// TIA Portal project "FactoryIO_Template_S7-1200_V16_V16" (V16)
// Vorlageprojekt für das Buch mit Zielsystem S7-1200

(* hardware
DEVICE "S7-1200-Station_1"  S7-1200 Station
   slot 0: "Baugruppenträger_0"  Rack  V1.0
   slot 1: "PLC_1"  CPU 1211C DC/DC/DC  6ES7 211-1AE40-0XB0  V4.1
*)

// ===== PLC "PLC_1"  CPU 1211C DC/DC/DC =====

VAR_GLOBAL   // PLC tag table "Standard-Variablentabelle"
   "fill valve" AT %A0.0 : Bool;
   "start" AT %E0.0 : Bool;
   "stop" AT %E0.1 : Bool;
   "Tag_4" AT %I10.0 : Bool;
   "Tag_5" AT %Q10.0 : Bool;
   "Tag_6" AT %I10.1 : Bool;
   "x" AT %M0.0 : Bool;
   "conveyor" AT %Q0.1 : Bool;
   "t1(1)" AT %M0.1 : Bool;
   "axis sensor" AT %I0.3 : Bool;
   "n" AT %M0.2 : Bool;
   "two axis pick and place 1 z" AT %Q0.2 : Bool;
   "diffuse sensor(1)" AT %I0.2 : Bool;
   "t2(1)" AT %M0.3 : Bool;
   "t2(2)" AT %M0.4 : Bool;
   "tank discharge" AT %Q0.3 : Bool;
   "Tag_1" AT %M0.5 : Bool;
   "t3(1)" AT %M0.6 : Bool;
   "n edge" AT %M0.7 : Bool;
   "t4(1)" AT %M1.0 : Bool;
END_VAR

// folder: System blocks/Program resources

DATA_BLOCK "T1"   // DB1
{ S7_Optimized_Access := 'TRUE' }
AUTHOR : Simatic
FAMILY : IEC
NAME : IEC_TMR
VERSION : 1.0
// stored: InstanceOfName IEC_TIMER
"IEC_TIMER"
BEGIN
END_DATA_BLOCK

DATA_BLOCK "T2"   // DB2
{ S7_Optimized_Access := 'TRUE' }
AUTHOR : Simatic
FAMILY : IEC
NAME : IEC_TMR
VERSION : 1.0
// stored: InstanceOfName IEC_TIMER
"IEC_TIMER"
BEGIN
END_DATA_BLOCK

DATA_BLOCK "T3"   // DB3
{ S7_Optimized_Access := 'TRUE' }
AUTHOR : Simatic
FAMILY : IEC
NAME : IEC_TMR
VERSION : 1.0
// stored: InstanceOfName IEC_TIMER
"IEC_TIMER"
BEGIN
END_DATA_BLOCK

DATA_BLOCK "T4"   // DB4
{ S7_Optimized_Access := 'TRUE' }
AUTHOR : Simatic
FAMILY : IEC
NAME : IEC_TMR
VERSION : 1.0
// stored: InstanceOfName IEC_TIMER
"IEC_TIMER"
BEGIN
END_DATA_BLOCK

// folder: (top level)

FUNCTION "MHJ-PLC-Lab-Function-S71200" : Void   // FC9000, SCL
{ S7_Optimized_Access := 'TRUE' }
VERSION : 0.1
   VAR_TEMP
      rdTimeReturn : Int;
      outputTime : DTL;
      SyncVal : Byte;
      forVal : Int;
      forVal_2 : Int;
      Value : Byte;
   END_VAR
   VAR CONSTANT
      CompVal : Byte := 16#34;
      Value_01 : Byte := 16#11;
      Value_01_DW : DWord := 16#A165_D992;
      Value_02_DW : DWord := 16#58BE_4401;
   END_VAR
BEGIN

   #Value:=PEEK(area := 16#82,
        dbNumber := 0,
        byteOffset := 511);
   #Value := #Value + 1;

   POKE(area := 16#82,
        dbNumber := 0,
        byteOffset := 511,
        value := #Value);

   POKE(area:=16#81,
        dbNumber:=0,
        byteOffset:=1016,
        value:=#Value_01_DW);
   POKE(area := 16#81,
        dbNumber := 0,
        byteOffset := 1020,
        value := #Value_02_DW);

   POKE(area := 16#81,
        dbNumber := 0,
        byteOffset := 511,
        value := B#16#00);

   FOR #forVal := 0 TO 120 DO
       FOR #forVal_2:=0 TO 10 DO
           #rdTimeReturn:=RD_SYS_T(#outputTime);
           #rdTimeReturn := WR_SYS_T(#outputTime);
           #rdTimeReturn := RD_SYS_T(#outputTime);
           #rdTimeReturn := WR_SYS_T(#outputTime);
       END_FOR;
       #SyncVal:= PEEK(area := 16#81,
                      dbNumber := 0,
                      byteOffset := 511);
       IF #SyncVal = #CompVal THEN
          GOTO M_1;
       END_IF;
   END_FOR;
   RETURN;

   M_1:
   POKE(area := 16#81,
        dbNumber := 0,
        byteOffset := 511,
        value := B#16#0);
END_FUNCTION

ORGANIZATION_BLOCK "Main"   // OB1, LAD, ProgramCycle
TITLE = "Main Program Sweep (Cycle)"
{ S7_Optimized_Access := 'TRUE' }
VERSION : 0.1
   VAR_INPUT
      Initial_Call : Bool;   // Initial call of this OB
      Remanence : Bool;   // =True, if remanent data are available
   END_VAR
   VAR_TEMP   // added for the SCL form of the ladder/FBD networks
      _w1 : Bool;
   END_VAR
BEGIN

REGION Network 1: Konnektierungsbaustein für PLC-Lab
   // Im Netzwerk 1 wird der Konnektierungsbaustein für PLC-Lab aufgerufen.
   // Dieser Aufruf darf nicht entfernt werden!
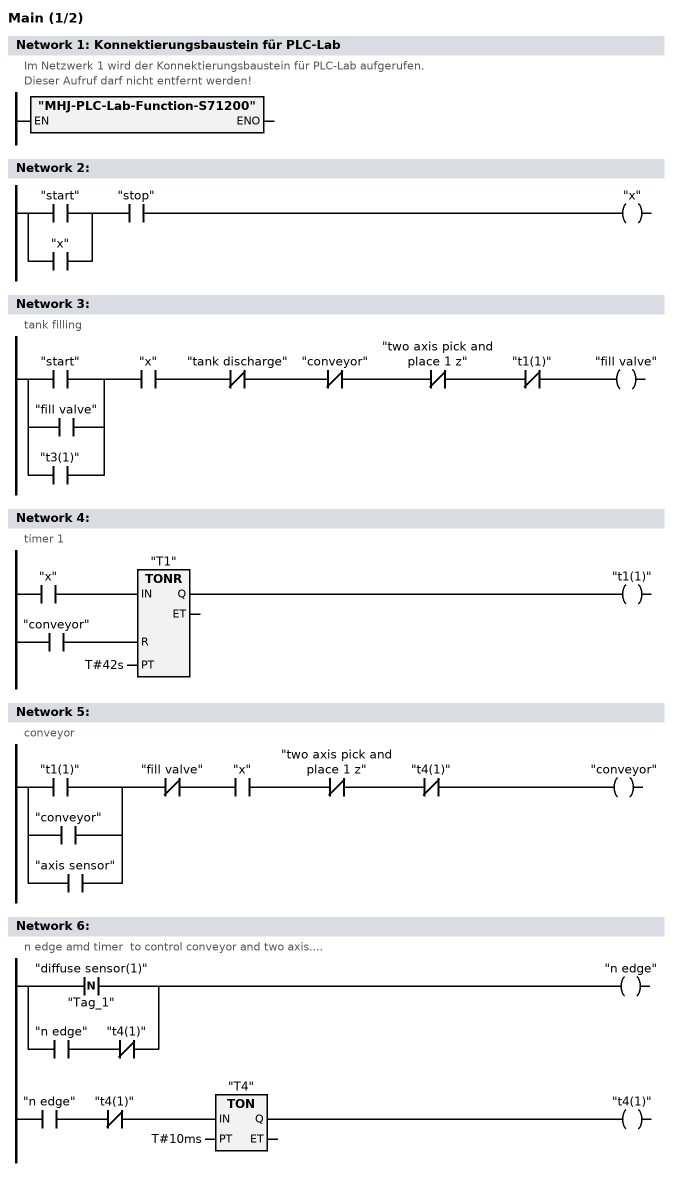
   RUNG wire#powerrail
      "MHJ-PLC-Lab-Function-S71200"()
   END_RUNG
   // the same network as SCL:
   "MHJ-PLC-Lab-Function-S71200"();
END_REGION

REGION Network 2
   RUNG wire#powerrail
      Contact( "start" )
      wire#w1
      Contact( "stop" )
      Coil( "x" )
   END_RUNG
   RUNG wire#powerrail
      Contact( "x" )
   END_RUNG wire#w1
   // the same network as SCL:
   "x" := ("start" OR "x") AND "stop";
END_REGION

REGION Network 3
   // tank filling
   RUNG wire#powerrail
      Contact( "start" )
      wire#w1
      Contact( "x" )
      I_Contact( "tank discharge" )
      I_Contact( "conveyor" )
      I_Contact( "two axis pick and place 1 z" )
      I_Contact( "t1(1)" )
      Coil( "fill valve" )
   END_RUNG
   RUNG wire#powerrail
      Contact( "fill valve" )
   END_RUNG wire#w1
   RUNG wire#powerrail
      Contact( "t3(1)" )
   END_RUNG wire#w1
   // the same network as SCL:
   "fill valve" := ("start" OR "fill valve" OR "t3(1)") AND "x" AND NOT "tank discharge" AND NOT "conveyor" AND NOT "two axis pick and place 1 z" AND NOT "t1(1)";
END_REGION

REGION Network 4
   // timer 1
   "T1".TONR(IN := "x", R := "conveyor", PT := T#42s);
   "t1(1)" := "T1".Q;
END_REGION

REGION Network 5
   // conveyor
   RUNG wire#powerrail
      Contact( "t1(1)" )
      wire#w1
      I_Contact( "fill valve" )
      Contact( "x" )
      I_Contact( "two axis pick and place 1 z" )
      I_Contact( "t4(1)" )
      Coil( "conveyor" )
   END_RUNG
   RUNG wire#powerrail
      Contact( "conveyor" )
   END_RUNG wire#w1
   RUNG wire#powerrail
      Contact( "axis sensor" )
   END_RUNG wire#w1
   // the same network as SCL:
   "conveyor" := ("t1(1)" OR "conveyor" OR "axis sensor") AND NOT "fill valve" AND "x" AND NOT "two axis pick and place 1 z" AND NOT "t4(1)";
END_REGION

REGION Network 6
   // n edge amd timer  to control conveyor and two axis....
   #_w1 := NOT "diffuse sensor(1)" AND "Tag_1";   // falling edge of "diffuse sensor(1)"
   "Tag_1" := "diffuse sensor(1)";
   "n edge" := #_w1 OR ("n edge" AND NOT "t4(1)");
   "T4".TON(IN := "n edge" AND NOT "t4(1)", PT := T#10ms);
   "t4(1)" := "T4".Q;
END_REGION

REGION Network 7
   // two axis acuator
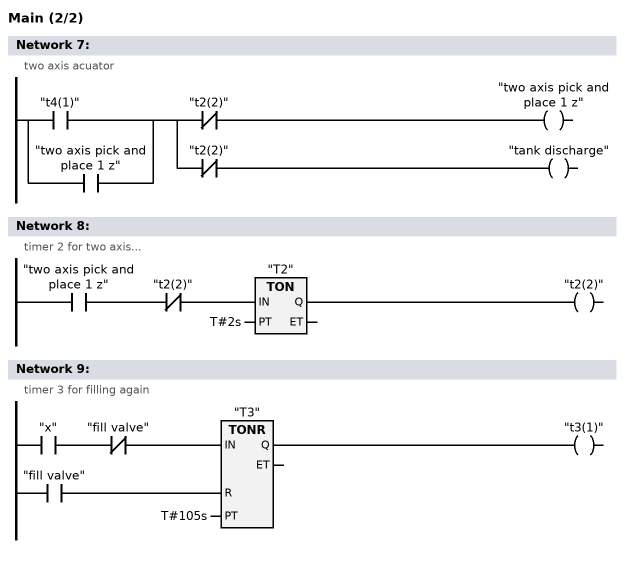
   RUNG wire#powerrail
      Contact( "t4(1)" )
      wire#w1
      I_Contact( "t2(2)" )
      Coil( "two axis pick and place 1 z" )
   END_RUNG
   RUNG wire#powerrail
      Contact( "two axis pick and place 1 z" )
   END_RUNG wire#w1
   RUNG wire#w1
      I_Contact( "t2(2)" )
      Coil( "tank discharge" )
   END_RUNG
   // the same network as SCL:
   #_w1 := "t4(1)" OR "two axis pick and place 1 z";
   "two axis pick and place 1 z" := #_w1 AND NOT "t2(2)";
   "tank discharge" := #_w1 AND NOT "t2(2)";
END_REGION

REGION Network 8
   // timer 2 for two axis...
   "T2".TON(IN := "two axis pick and place 1 z" AND NOT "t2(2)", PT := T#2s);
   "t2(2)" := "T2".Q;
END_REGION

REGION Network 9
   // timer 3 for filling again
   "T3".TONR(IN := "x" AND NOT "fill valve", R := "fill valve", PT := T#105s);
   "t3(1)" := "T3".Q;
END_REGION
END_ORGANIZATION_BLOCK